TYPE PB_64Byte :
STRUCT
	Header 		: BYTE;
	DATA 		: ARRAY[0..8] OF PB_Dateneintrag;
END_STRUCT
END_TYPE

(* stored: Version 1.1.0.1, ProductVersion 3.1.4024.9
   DUT PB_64Byte: Id {5d40b918-b839-4b71-a5e1-cdef0aca18c9} *)
